INTERFACE IF_EmptyRegister EXTENDS __SYSTEM.IQueryInterface

METHOD Get : DINT
VAR_INPUT
END_VAR
END_METHOD

PROPERTY xReadyForGet : BOOL
GET
END_GET
END_PROPERTY

END_INTERFACE

(* stored: Version 1.1.0.1
   Itf IF_EmptyRegister: Id {95e70f9b-8d68-4249-9198-0a0b867ca004}
   Method Get: Id {f697f8d1-dd29-4f8d-9a39-d29fb7ca472f}
   Property xReadyForGet: Id {ab3a0d7e-a581-4982-a2fd-c59ae6ac3e3c}
   Get Get: Id {8802ca4c-3526-4d62-9882-93cca422cfd8} *)
